FUNCTION_BLOCK FB_BarcodeInspection
VAR_INPUT
	bEnable				: BOOL;
	bTrigger			: BOOL;
	bBypassFGHS			: BOOL;
	bBarcodeGood		: ARRAY [1..4] OF BOOL;
	bBarcodeBad			: ARRAY [1..4] OF BOOL;
	bDoneRead			: ARRAY [1..4] OF BOOL;
	BarcodeData1		: STRING;
	BarcodeData2		: STRING;
	BarcodeData3		: STRING;
	BarcodeData4		: STRING;
	bPalletReady		: ARRAY [1..4] OF BOOL;
	bResetCounter		: BOOL;
END_VAR
VAR_OUTPUT
	bBarcodeChecked		: BOOL;
	BarcodeResult		: STRING;
	iPlacingLine		: INT;
	bReject				: BOOL;
	bProductFound		: ARRAY [1..4] OF BOOL;
	RejectID			: INT;
	RejectMsg			: STRING;
END_VAR
VAR_OUTPUT PERSISTENT
	CountReject			: UINT;
END_VAR
VAR_IN_OUT
	ar_ProductInfo		: ARRAY [1..4] OF stProductInfo;
	PlannedEAN			: ARRAY [1..4] OF STRING;
	PlannedCodeVariant	: ARRAY [1..4] OF STRING;
END_VAR
VAR
	Sequence			: INT;
	DoneCheck			: BOOL;
	BarcodeEAN			: STRING;
	CodeVariant			: STRING;
	BarcodeLinkUp		: STRING;
	TimeOut				: TON;
	NotFound			: BOOL;
	i					: INT;
	Index				: INT;
	plaintext: INT;
END_VAR


IF bResetCounter THEN // Jika bResetCounter aktif
	CountReject := 0; // Set ulang CountReject menjadi 0
END_IF // Selesai kondisi IF

IF bEnable THEN // Jika bEnable aktif
	
	(*----Check Barcode -----*)
	CASE Sequence OF // Pemilihan kasus berdasarkan nilai Sequence
		0:	
			IF bTrigger THEN // Jika bTrigger aktif
				DoneCheck		:= FALSE; // Set DoneCheck menjadi tidak aktif
				bBarcodeChecked	:= FALSE; // Set bBarcodeChecked menjadi tidak aktif
				bReject			:= FALSE; // Set bReject menjadi tidak aktif
				iPlacingLine	:= 0; // Set iPlacingLine menjadi 0
				RejectID		:= 0; // Set RejectID menjadi 0
				RejectMsg		:= ''; // Set RejectMsg menjadi string kosong
				BarcodeResult	:= ''; // Set BarcodeResult menjadi string kosong
				BarcodeEAN		:= ''; // Set BarcodeEAN menjadi string kosong
				CodeVariant		:= ''; // Set CodeVariant menjadi string kosong
				BarcodeLinkUp	:= ''; // Set BarcodeLinkUp menjadi string kosong
				Sequence		:= 10; // Ganti nilai Sequence menjadi 10
			END_IF // Selesai kondisi IF
			
		10:
			TimeOut(IN:=TRUE, PT:=T#5S); // Aktifkan TimeOut dengan periode 5 detik
			IF bBarcodeGood[1] AND bDoneRead[1] THEN // Jika bBarcodeGood[1] aktif dan bDoneRead[1] aktif
				BarcodeResult 	:= BarcodeData1; // Set BarcodeResult dari BarcodeData1
				Sequence		:= 11; // Ganti nilai Sequence menjadi 11
			ELSIF bBarcodeGood[2] AND bDoneRead[2] THEN // Jika bBarcodeGood[2] aktif dan bDoneRead[2] aktif
				BarcodeResult 	:= BarcodeData2; // Set BarcodeResult dari BarcodeData2
				Sequence		:= 11; // Ganti nilai Sequence menjadi 11
			ELSIF bBarcodeGood[3] AND bDoneRead[3] THEN // Jika bBarcodeGood[3] aktif dan bDoneRead[3] aktif
				BarcodeResult 	:= BarcodeData3; // Set BarcodeResult dari BarcodeData3
				Sequence		:= 11; // Ganti nilai Sequence menjadi 11
			ELSIF bBarcodeGood[4] AND bDoneRead[4] THEN // Jika bBarcodeGood[4] aktif dan bDoneRead[4] aktif
				BarcodeResult 	:= BarcodeData4; // Set BarcodeResult dari BarcodeData4
				Sequence		:= 11; // Ganti nilai Sequence menjadi 11
			ELSIF (bBarcodeBad[1] AND bBarcodeBad[2] AND bBarcodeBad[3] AND bBarcodeBad[4]) OR TimeOut.Q THEN // Jika semua bBarcodeBad aktif atau TimeOut tercapai
				TimeOut(IN:=FALSE); // Nonaktifkan TimeOut
				RejectID		:= 1; // Set RejectID menjadi 1
				RejectMsg		:= 'Reject Bad Read Barcode'; // Set RejectMsg
				Sequence		:= 999; // Ganti nilai Sequence menjadi 999
			END_IF // Selesai kondisi IF
			
		11:	(* Split Barcode *)
			BarcodeEAN		:= DELETE(DELETE(BarcodeResult,3,0),24,15); // Ambil bagian tertentu dari BarcodeResult sebagai BarcodeEAN
			CodeVariant		:= DELETE(DELETE(BarcodeResult,19,0),20,3); // Ambil bagian tertentu dari BarcodeResult sebagai CodeVariant
			BarcodeLinkUp	:= DELETE(DELETE(BarcodeResult,33,0),6,3); // Ambil bagian tertentu dari BarcodeResult sebagai BarcodeLinkUp
			Sequence		:= 12; // Ganti nilai Sequence menjadi 12
			
		12: (* Check EAN *)
			FOR i := 1 TO 4 BY 1 DO // Loop untuk setiap elemen PlannedEAN
				IF PlannedEAN[i] <> '' AND BarcodeEAN = PlannedEAN[i] AND PlannedEAN[i] <> ar_ProductInfo[i].EANVariant THEN // Jika PlannedEAN tidak kosong dan BarcodeEAN sama dengan PlannedEAN dan PlannedEAN tidak sama dengan ar_ProductInfo[i].EANVariant
					ar_ProductInfo[i].EANVariant	:= PlannedEAN[i]; // Update nilai ar_ProductInfo[i].EANVariant
					bProductFound[i]				:= TRUE; // Set bProductFound[i] menjadi TRUE
					Sequence						:= 20; // Ganti nilai Sequence menjadi 20
					EXIT; // Keluar dari loop FOR
				END_IF // Selesai kondisi IF
			END_FOR // Selesai loop FOR
			
			IF i > 4 THEN // Jika i melebihi 4
				i 				:= 0; // Set i menjadi 0
				Sequence		:= 20; // Ganti nilai Sequence menjadi 20
			END_IF // Selesai kondisi IF
			
		20:	
			FOR i := 1 TO 4 BY 1 DO // Loop untuk setiap elemen ar_ProductInfo
				IF BarcodeLinkUp = ar_ProductInfo[i].LinkUpSource  AND BarcodeEAN = ar_ProductInfo[i].EANVariant THEN // Jika BarcodeLinkUp sama dengan ar_ProductInfo[i].LinkUpSource dan BarcodeEAN sama dengan ar_ProductInfo[i].EANVariant
					iPlacingLine	 		:= i; // Set iPlacingLine
					Sequence				:= 21; // Ganti nilai Sequence menjadi 21
					EXIT; // Keluar dari loop FOR
				END_IF; // Selesai kondisi IF
			END_FOR; // Selesai loop FOR	
			IF i > 4 THEN // Jika i melebihi 4
				bBarcodeChecked	:= FALSE; // Set bBarcodeChecked menjadi FALSE
				NotFound		:= TRUE; // Set NotFound menjadi TRUE
				RejectID		:= 2; // Set RejectID menjadi 2
				RejectMsg		:= 'Barcode Result Not Matched Any References'; // Set RejectMsg
				Sequence		:= 999; // Ganti nilai Sequence menjadi 999
			END_IF; // Selesai kondisi IF
			
		21:
			IF CodeVariant <> ar_ProductInfo[iPlacingLine].CodeVariant THEN // Jika CodeVariant tidak sama dengan ar_ProductInfo[iPlacingLine].CodeVariant
				ar_ProductInfo[iPlacingLine].CodeVariant	:= CodeVariant; // Update nilai ar_ProductInfo[iPlacingLine].CodeVariant
				bProductFound[iPlacingLine

]					:= TRUE; // Set bProductFound[iPlacingLine] menjadi TRUE
				Sequence									:= 30; // Ganti nilai Sequence menjadi 30
			ELSE
				Sequence									:= 30; // Ganti nilai Sequence menjadi 30
			END_IF
			
		30:
			IF bPalletReady[iPlacingLine] THEN // Jika bPalletReady[iPlacingLine] aktif
				TimeOut(IN:=FALSE); // Nonaktifkan TimeOut
				bBarcodeChecked	:=	TRUE; // Set bBarcodeChecked menjadi TRUE
				Sequence		:=	1000;	// Ganti nilai Sequence menjadi 1000	
			ELSE
				TimeOut(IN:=TRUE, PT:=T#30S); // Aktifkan TimeOut dengan periode 30 detik
				IF TimeOut.Q THEN // Jika TimeOut tercapai
				TimeOut(IN:=FALSE); // Nonaktifkan TimeOut
				RejectID		:= 3; // Set RejectID menjadi 3
				RejectMsg		:= 'Reject Placing Not Ready'; // Set RejectMsg
				Sequence		:= 999; // Ganti nilai Sequence menjadi 999
				END_IF
			END_IF
			
		999:
			TimeOut(IN:=FALSE); // Nonaktifkan TimeOut
			iPlacingLine	:= 0; // Set iPlacingLine menjadi 0
			bBarcodeChecked	:=	TRUE; // Set bBarcodeChecked menjadi TRUE
			bReject 		:=	TRUE; // Set bReject menjadi TRUE
			CountReject		:= 	CountReject + 1; // Tambahkan 1 pada CountReject
			Sequence		:=	1000;	// Ganti nilai Sequence menjadi 1000	
	
		1000:
			DoneCheck	:= TRUE; // Set DoneCheck menjadi TRUE
			IF NOT bTrigger THEN // Jika bTrigger tidak aktif
				bProductFound[1]	:= FALSE;	// Set bProductFound[1] menjadi FALSE
				bProductFound[2]	:= FALSE; // Set bProductFound[2] menjadi FALSE
				bProductFound[3]	:= FALSE; // Set bProductFound[3] menjadi FALSE
				bProductFound[4]	:= FALSE; // Set bProductFound[4] menjadi FALSE
				NotFound			:= FALSE; // Set NotFound menjadi FALSE
				bBarcodeChecked		:= FALSE; // Set bBarcodeChecked menjadi FALSE
				bReject				:= FALSE; // Set bReject menjadi FALSE
				Sequence			:= 0; // Ganti nilai Sequence menjadi 0
			END_IF // Selesai kondisi IF
			
	END_CASE // Selesai pemilihan kasus
	
ELSE
	TimeOut(IN:=FALSE); // Nonaktifkan TimeOut
	NotFound			:= FALSE; // Set NotFound menjadi FALSE
	bBarcodeChecked		:= FALSE; // Set bBarcodeChecked menjadi FALSE
	bReject				:= FALSE; // Set bReject menjadi FALSE
	Sequence			:= 0; // Ganti nilai Sequence menjadi 0
	iPlacingLine		:= 0; // Set iPlacingLine menjadi 0
	i					:= 0; // Set i menjadi 0
END_IF // Selesai kondisi IF

END_FUNCTION_BLOCK

(* stored: Version 1.1.0.1, ProductVersion 3.1.4024.6
   POU FB_BarcodeInspection: Id {30941f97-6106-4e76-9db7-8cb51e5c6809}, SpecialFunc None *)
